(*

.. <legal notes>

legal notes
=================
| SPDX-FileCopyrightText: © 2025 Oleksandr Tiutyk <trofimich@gmail.com>
| SPDX-License-Identifier: LGPL-3.0-only
| For details check: LGPL-3.0-only_

.. _LGPL-3.0-only: https://www.gnu.org/licenses/lgpl-3.0.en.html

.. </legal notes>

*)

FUNCTION_BLOCK SignalControlledIntersectionAutomationRunner EXTENDS TOF_AutomationEngine.AutomationRunner<1>
VAR_OUTPUT
	SignalControlledIntersectionAutomationController : SignalControlledIntersectionAutomationController(THIS^);
END_VAR
VAR
	_ClassName : STRING := __POUNAME();
	
	_AutomationControllers : ARRAY [0..0] OF TOF_AutomationEngine.IAutomationController := [SignalControlledIntersectionAutomationController];
END_VAR

{attribute 'monitoring' := 'call'}
PROPERTY AutomationUnits : REFERENCE TO ARRAY [0.._AutomationUnitCount - 1] OF TOF_AutomationEngine.IAutomationController
GET
AutomationUnits REF= _AutomationControllers;
END_GET
END_PROPERTY

{attribute 'monitoring' := 'call'}
PROPERTY ClassName : STRING
GET
ClassName := _ClassName;
END_GET
END_PROPERTY

//FB_Init is always available implicitly and it is used primarily for initialization.
//The return value is not evaluated. For a specific influence, you can also declare the
//methods explicitly and provide additional code there with the standard initialization
//code. You can evaluate the return value.
METHOD FB_Init: BOOL
VAR_INPUT
    bInitRetains: BOOL; // TRUE: the retain variables are initialized (reset warm / reset cold)
    bInCopyCode: BOOL;  // TRUE: the instance will be copied to the copy code afterward (online change)   
END_VAR
TrySetSimulationMode(TRUE);
END_METHOD

{attribute 'monitoring' := 'call'}
PROPERTY Size : ULINT
GET
Size := XSIZEOF(THIS^);
END_GET
END_PROPERTY

END_FUNCTION_BLOCK

(* stored: Version 1.1.0.1
   POU SignalControlledIntersectionAutomationRunner: Id {ff964406-6e7d-46be-9bc3-ae0ec1a8df3e}, SpecialFunc None
   Property AutomationUnits: Id {6362bba8-7b43-445e-977a-8defd358fba7}
   Get Get: Id {fccbb52a-40a3-46d6-904d-074ece3ee424}
   Property ClassName: Id {44015b9d-a297-4fcc-8765-1882288ab888}
   Get Get: Id {cab8ddbf-0d31-4c51-ad36-9a0a06b1f991}
   Method FB_Init: Id {9c8ff6ec-3304-47ad-8fa3-9fc9a9937959}
   Property Size: Id {23eac530-e293-442f-b701-6a55d41e89b4}
   Get Get: Id {6b2e6577-47f6-43bc-b255-c7867b3833f7} *)
